(* CoDeSys 2.3.5.6 project: szlendak_03_fbd.pro *)
(* Libraries: Standard.lib*4.1.15 17:23:13, SYSLIBCALLBACK.LIB*4.1.15 17:23:13 *)

(* PLC configuration (modules and I/O channels)
I1 AT %IX0.0 [LocalBitInput] Input I1
I2 AT %IX0.1 [LocalBitInput] Input I2
I3 AT %IX0.2 [LocalBitInput] Input I3
I4 AT %IX0.3 [LocalBitInput] Input I4
I5 AT %IX0.4 [LocalBitInput] Input I5
I6 AT %IX0.5 [LocalBitInput] Input I6
I7 AT %IX0.6 [LocalBitInput] Input I7
I8 AT %IX0.7 [LocalBitInput] Input I8
I9 AT %IX1.0 [LocalBitInput] Input I9
I10 AT %IX1.1 [LocalBitInput] Input I10
I11 AT %IX1.2 [LocalBitInput] Input I11
I12 AT %IX1.3 [LocalBitInput] Input I12
I13 AT %IX1.4 [LocalDiagInput] Diagnostic Input I13
I14 AT %IX1.5 [LocalDiagInput] Diagnostic Input I14
I15 AT %IX1.6 [LocalDiagInput] Diagnostic Input I15
I16 AT %IX1.7 [LocalDiagInput] Diagnostic Input I16
I7_Analog AT %IW2 [LocalAnalogIn] Input I7, 10Bit, 0-10VDC
I8_Analog AT %IW4 [LocalAnalogIn] Input I8, 10Bit, 0-10VDC
I11_Analog AT %IW6 [LocalAnalogIn] Input I11, 10Bit, 0-10VDC
I12_Analog AT %IW8 [LocalAnalogIn] Input I12, 10Bit, 0-10VDC
Q1 AT %QX0.0 [LocalBitOutput] Transistor-Output Q1
Q2 AT %QX0.1 [LocalBitOutput] Transistor-Output Q2
Q3 AT %QX0.2 [LocalBitOutput] Transistor-Output Q3
Q4 AT %QX0.3 [LocalBitOutput] Transistor-Output Q4
Q5 AT %QX0.4 [LocalBitOutput] Transistor-Output Q5
Q6 AT %QX0.5 [LocalBitOutput] Transistor-Output Q6
Q7 AT %QX0.6 [LocalBitOutput] Transistor-Output Q7
Q8 AT %QX0.7 [LocalBitOutput] Transistor-Output Q8
No Analog Output [EC4P_NoAnalogOutput] node 1, in %IB10 out %QB1
No Keys [EC4P_NoKeys] node 2, in %IB10 out %QB1
No Counter [EC4P_NoCounter] node 3, in %IB10 out %QB1
No Extension [EC4P_NoExtension] node 0, in %IB10 out %QB1
*)

(* Global variable list: Zmienne_globalne *)
VAR_GLOBAL
	jest1: BOOL;
	jest2: BOOL;
	jest3: BOOL;
	jest4: BOOL;
	jest5: BOOL;
	jest6: BOOL;
	jest7: BOOL;
	jest8: BOOL;
	jest9: BOOL;
	jest0: BOOL;
	wartosc: INT;
	RESET: BOOL;
	LICZNIK1: CTU;
	T1: TON;
	T2: TON;
	TT1: TIME;
	TT2: TIME;
	Q12: BOOL;
	W1: BOOL;
END_VAR

(* POU PLC_PRG, FBD *)
PROGRAM PLC_PRG
VAR
 Q9:BOOL;
 Q10:BOOL;
END_VAR
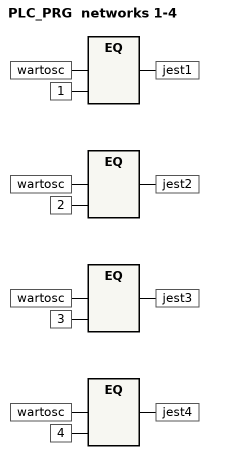
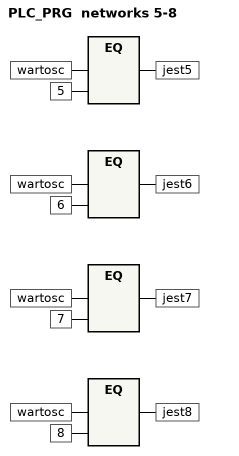
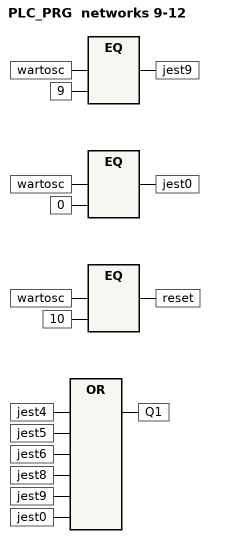
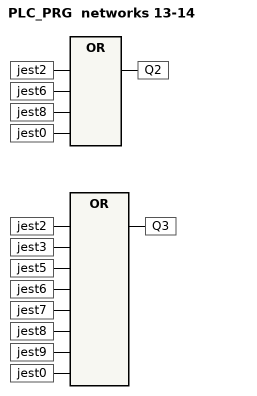
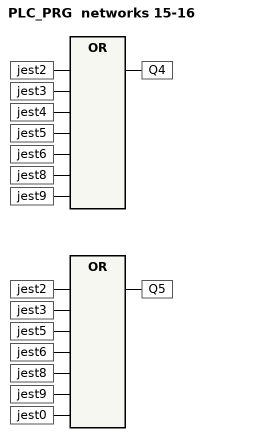
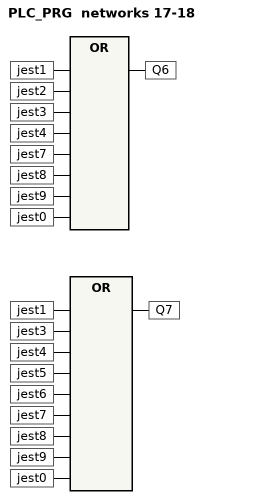
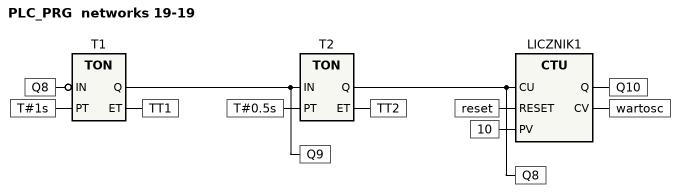
_FBD_ (* Function Block Diagram *)
NETWORK 1
	EQ(wartosc, 1) => jest1
NETWORK 2
	EQ(wartosc, 2) => jest2
NETWORK 3
	EQ(wartosc, 3) => jest3
NETWORK 4
	EQ(wartosc, 4) => jest4
NETWORK 5
	EQ(wartosc, 5) => jest5
NETWORK 6
	EQ(wartosc, 6) => jest6
NETWORK 7
	EQ(wartosc, 7) => jest7
NETWORK 8
	EQ(wartosc, 8) => jest8
NETWORK 9
	EQ(wartosc, 9) => jest9
NETWORK 10
	EQ(wartosc, 0) => jest0
NETWORK 11
	EQ(wartosc, 10) => reset
NETWORK 12
	OR(jest4, jest5, jest6, jest8, jest9, jest0) => Q1
NETWORK 13
	OR(jest2, jest6, jest8, jest0) => Q2
NETWORK 14
	OR(jest2, jest3, jest5, jest6, jest7, jest8, jest9, jest0) => Q3
NETWORK 15
	OR(jest2, jest3, jest4, jest5, jest6, jest8, jest9) => Q4
NETWORK 16
	OR(jest2, jest3, jest5, jest6, jest8, jest9, jest0) => Q5
NETWORK 17
	OR(jest1, jest2, jest3, jest4, jest7, jest8, jest9, jest0) => Q6
NETWORK 18
	OR(jest1, jest3, jest4, jest5, jest6, jest7, jest8, jest9, jest0) => Q7
NETWORK 19
	LICZNIK1:CTU(CU: <T2:TON(IN: <T1:TON(IN: NOT Q8, PT: T#1s, ET => TT1) => Q9>, PT: T#0.5s, ET => TT2) => Q8>, RESET: reset, PV: 10, CV => wartosc) => Q10
_END_FBD_
(* the same logic as Structured Text *)
(* Network 1 *)
jest1 := wartosc = 1;
(* Network 2 *)
jest2 := wartosc = 2;
(* Network 3 *)
jest3 := wartosc = 3;
(* Network 4 *)
jest4 := wartosc = 4;
(* Network 5 *)
jest5 := wartosc = 5;
(* Network 6 *)
jest6 := wartosc = 6;
(* Network 7 *)
jest7 := wartosc = 7;
(* Network 8 *)
jest8 := wartosc = 8;
(* Network 9 *)
jest9 := wartosc = 9;
(* Network 10 *)
jest0 := wartosc = 0;
(* Network 11 *)
reset := wartosc = 10;
(* Network 12 *)
Q1 := jest4 OR jest5 OR jest6 OR jest8 OR jest9 OR jest0;
(* Network 13 *)
Q2 := jest2 OR jest6 OR jest8 OR jest0;
(* Network 14 *)
Q3 := jest2 OR jest3 OR jest5 OR jest6 OR jest7 OR jest8 OR jest9 OR jest0;
(* Network 15 *)
Q4 := jest2 OR jest3 OR jest4 OR jest5 OR jest6 OR jest8 OR jest9;
(* Network 16 *)
Q5 := jest2 OR jest3 OR jest5 OR jest6 OR jest8 OR jest9 OR jest0;
(* Network 17 *)
Q6 := jest1 OR jest2 OR jest3 OR jest4 OR jest7 OR jest8 OR jest9 OR jest0;
(* Network 18 *)
Q7 := jest1 OR jest3 OR jest4 OR jest5 OR jest6 OR jest7 OR jest8 OR jest9 OR jest0;
(* Network 19 *)
T1(IN := NOT Q8, PT := T#1s);
TT1 := T1.ET;
Q9 := T1.Q;
T2(IN := T1.Q, PT := T#0.5s);
TT2 := T2.ET;
Q8 := T2.Q;
LICZNIK1(CU := T2.Q, RESET := reset, PV := 10);
wartosc := LICZNIK1.CV;
Q10 := LICZNIK1.Q;
END_PROGRAM
